TYPE "MEStoPLC_RecipeParameter_OP220"
VERSION : 0.1
   STRUCT
      Press { S7_SetPoint := 'False'} : "PresserRecipe";
      ATEQ : "ATEQRecipe";
   END_STRUCT;

END_TYPE

